// TwinCAT 3 PLC project PLC_UU_V01
// ProgramVersion: 3.1.4022.4
// libraries:
//   Tc2_MC2, * (Beckhoff Automation GmbH)
//   Tc2_Standard, * (Beckhoff Automation GmbH)
//   Tc2_System, * (Beckhoff Automation GmbH)
//   Tc3_Module, * (Beckhoff Automation GmbH)
//   VisuDialogs, * (System)
// project tree:
//   DUTs/ ST_AxisIn.TcDUT, ST_AxisInterface.TcDUT, ST_AxisOut.TcDUT, ST_Demo.TcDUT
//   / GlobalTextList.TcGTLO, PlcTask.TcTTO, Visualization Manager.TcVMO (not stored)
//   GVLs/ GVL_IO.TcGVL, GVL_Servo.TcGVL
//   POUs/ FB_Motion.TcPOU, MAIN.TcPOU, PRG_Servo1.TcPOU
//   VISUs/ TC_SERVO1.TcVIS

CONFIGURATION PLC_UU_V01
    RESOURCE PLC ON TwinCAT3
        TASK PlcTask(INTERVAL := T#10ms, PRIORITY := 20);
        PROGRAM MAIN WITH PlcTask : MAIN;
    END_RESOURCE
END_CONFIGURATION

// ---- DUTs/ST_AxisIn.TcDUT
TYPE ST_AxisIn :
STRUCT
	bEnable		: BOOL;
	fOverride	: LREAL;
	bManuelFw	: BOOL;
	bManuelBw	: BOOL;
	fVelocity	: LREAL;
	bMoveAbs	: BOOL;
	fPosition	: LREAL;
	bStop		:BOOL;
	bReset		:BOOL;

END_STRUCT
END_TYPE

// ---- DUTs/ST_AxisInterface.TcDUT
TYPE ST_AxisInterface :
STRUCT
	INPUT	: ST_AxisIn;
	OUTPUT	: ST_AxisOut;
	
END_STRUCT
END_TYPE

// ---- DUTs/ST_AxisOut.TcDUT
TYPE ST_AxisOut :
STRUCT
	bEnabled	: BOOL;
	bJogBusy	: BOOL;
	bJogDone	: BOOL;
	bMoveAbsDone: BOOL;
	bMoveAbsBusy: BOOL;
	bJogError	: BOOL;
	bPowerErr	: BOOL;
	bMoveAbsErr	: BOOL;
	bStopDone	: BOOL;
	bStopBusy	: BOOL;
	bStopErr	: BOOL;
	bStopActive : BOOL;	
	bResetDone	:BOOL;

END_STRUCT
END_TYPE

// ---- DUTs/ST_Demo.TcDUT
TYPE ST_Demo :
STRUCT
	bVar	: BOOL;
	sVar	: STRING;
	nVar	: INT;
	fVar	: LREAL;
	
END_STRUCT
END_TYPE

// ---- GVLs/GVL_IO.TcGVL
VAR_GLOBAL
	bInput1	AT%I*	: BOOL;
	bInput2	AT%I*	: BOOL;
	bInput3	AT%I*	: BOOL;
	bInput4	AT%I*	: BOOL;
	
	bOutput1	AT%Q*	: BOOL;
	bOutput2	AT%Q*	: BOOL;
	bOutput3	AT%Q*	: BOOL;
	bOutput4	AT%Q*	: BOOL;
	
	nInput1		AT%I*	: INT;
	nInput2		AT%I*	: INT;
	
	nOutput1	AT%Q*	: INT;
	nOutput2	AT%Q*	: INT;
	
END_VAR

// ---- GVLs/GVL_Servo.TcGVL
VAR_GLOBAL
	Axis1	: AXIS_REF;
	Axis2	: AXIS_REF;
	
	stAxis1	: ST_AxisInterface;
	stAxis2	: ST_AxisInterface;
	
	fbMotion1	: FB_Motion;
	fbMotion2	: FB_Motion;
	
END_VAR

// ---- POUs/MAIN.TcPOU
PROGRAM MAIN
VAR
	stDemo	: ST_Demo;
	stArrayDemo	: ARRAY[1..100]OF ST_Demo;
	
	i: INT;
	
END_VAR

IF bInput1	THEN
	FOR i:= 0 TO 100 DO
		stArrayDemo[i+1].nVar	:= i*i;
		stArrayDemo[i+1].fVar	:= INT_TO_LREAL(i)+1.345;
	END_FOR
END_IF

ACT_Motion();

PRG_Servo1();

ACTION ACT_Motion:
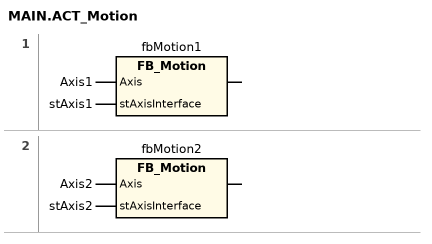
// NETWORK 1
fbMotion1(Axis := Axis1, stAxisInterface := stAxis1); // FB_Motion

// NETWORK 2
fbMotion2(Axis := Axis2, stAxisInterface := stAxis2); // FB_Motion
END_ACTION

END_PROGRAM

// ---- POUs/PRG_Servo1.TcPOU
PROGRAM PRG_Servo1
VAR
	nState: INT;
	bBaslat	: bool;
	bSensor1: BOOL;
	rSayici: R_TRIG;
	bSensor2: BOOL;
	nSayici: INT;
	nCounter: INT;
END_VAR

stAxis1.INPUT.bEnable	:= TRUE;
staxis1.INPUT.bStop:=FALSE;
stAxis1.INPUT.bReset := FALSE;


rSayici(CLK:= bSensor2, Q=> );
CASE nState OF
	
0:
	IF bBaslat AND staxis1.OUTPUT.bEnabled AND NOT stAxis1.OUTPUT.bPowerErr THEN
		nState	:= 10;
		nCounter := 0;
	END_IF
	
10:
	stAxis1.INPUT.bMoveAbs	:= TRUE;
	stAxis1.INPUT.fVelocity	:= 4000;
	stAxis1.INPUT.fPosition	:= 30000;
	
	IF stAxis1.OUTPUT.bMoveAbsBusy AND NOT stAxis1.OUTPUT.bMoveAbsErr THEN

		nState					:= 20;
		stAxis1.INPUT.bMoveAbs:=FALSE;

	ELSIF stAxis1.OUTPUT.bMoveAbsErr THEN
	
	nState					:= 999;
	nCounter := nState;
	stAxis1.INPUT.bMoveAbs	:= FALSE;

	END_IF
			
20:
	IF stAxis1.OUTPUT.bMoveAbsDone AND NOT stAxis1.OUTPUT.bMoveAbsErr THEN
		nState					:= 30;
		nCounter := nState;

	ELSIF stAxis1.OUTPUT.bMoveAbsErr THEN	
		nState					:= 999;
		nCounter := nState;

	END_IF
	
30:	
	IF bSensor1 THEN
		nState	:= 40;
		nCounter:=nState;
	END_IF
	
40:
	nCounter:=30;

	stAxis1.INPUT.bMoveAbs	:= TRUE;
	stAxis1.INPUT.fVelocity	:= 7000;
	stAxis1.INPUT.fPosition	:= 50000;
	
	IF stAxis1.OUTPUT.bMoveAbsBusy AND NOT stAxis1.OUTPUT.bMoveAbsErr THEN
		stAxis1.INPUT.bMoveAbs	:= FALSE;
		nState					:= 50;

	ELSIF stAxis1.OUTPUT.bMoveAbsErr THEN
		nState					:= 999;
		nCounter := nState;

		stAxis1.INPUT.bMoveAbs	:= FALSE;		
	END_IF
	
50:
	IF stAxis1.OUTPUT.bMoveAbsDone AND NOT stAxis1.OUTPUT.bMoveAbsErr THEN
		nState					:= 60;
		nCounter := nState;

	ELSIF stAxis1.OUTPUT.bMoveAbsErr THEN	
		nState					:= 999;
		nCounter := nState;

	END_IF

60:
	IF rSayici.Q AND nSayici<5 THEN
		nSayici	:= nSayici+1;	
	ELSIF nSayici>=5 THEN
		nSayici	:=0;
		nState	:= 70;
		nCounter := nState;
	END_IF

70:
	stAxis1.INPUT.bMoveAbs	:= TRUE;

	stAxis1.INPUT.fVelocity	:= 8000;
	stAxis1.INPUT.fPosition	:= 0;
	nCounter:=60;
	IF stAxis1.OUTPUT.bMoveAbsBusy AND NOT stAxis1.OUTPUT.bMoveAbsErr THEN
		stAxis1.INPUT.bMoveAbs	:= FALSE;
		nState					:= 80;
		nCounter := nState;

	ELSIF stAxis1.OUTPUT.bMoveAbsErr THEN
		nState					:= 999;
		nCounter := nState;

		stAxis1.INPUT.bMoveAbs	:= FALSE;		
	END_IF
	
80:
	IF stAxis1.OUTPUT.bMoveAbsDone AND NOT stAxis1.OUTPUT.bMoveAbsErr THEN
				nState	:= 0;
				nCounter := nState;

	ELSIF stAxis1.OUTPUT.bMoveAbsErr THEN	
		nState					:= 999;
		nCounter := nState;

	END_IF
	
END_CASE

IF stAxis1.OUTPUT.bPowerErr THEN
	stAxis1.INPUT.bReset := TRUE;
	nState:=0;
END_IF

IF NOT bBaslat THEN
	
staxis1.INPUT.bStop:=TRUE;
stAxis1.INPUT.bMoveAbs	:= FALSE;
staxis1.OUTPUT.bEnabled:=TRUE;


		IF staxis1.OUTPUT.bEnabled
		AND NOT stAxis1.OUTPUT.bPowerErr 
		AND NOT stAxis1.OUTPUT.bMoveAbsErr
		AND NOT staxis1.OUTPUT.bStopErr 
		AND  staxis1.OUTPUT.bStopBusy THEN
	
	staxis1.INPUT.bStop:=FALSE;
	nState:=nCounter;

	END_IF

END_IF

END_PROGRAM

// ---- POUs/FB_Motion.TcPOU
FUNCTION_BLOCK FB_Motion
VAR_INPUT

	
END_VAR
VAR_OUTPUT
	
END_VAR
VAR
	fbMcPower	: MC_Power;
	fbMcJog: MC_Jog;
	fbMcMoveAbs: MC_MoveAbsolute;
	fbMcStop: MC_Stop;
	fbMcReset: MC_Reset;
END_VAR

VAR_IN_OUT
	Axis			: AXIS_REF;
	stAxisInterface	: ST_AxisInterface;
	
END_VAR

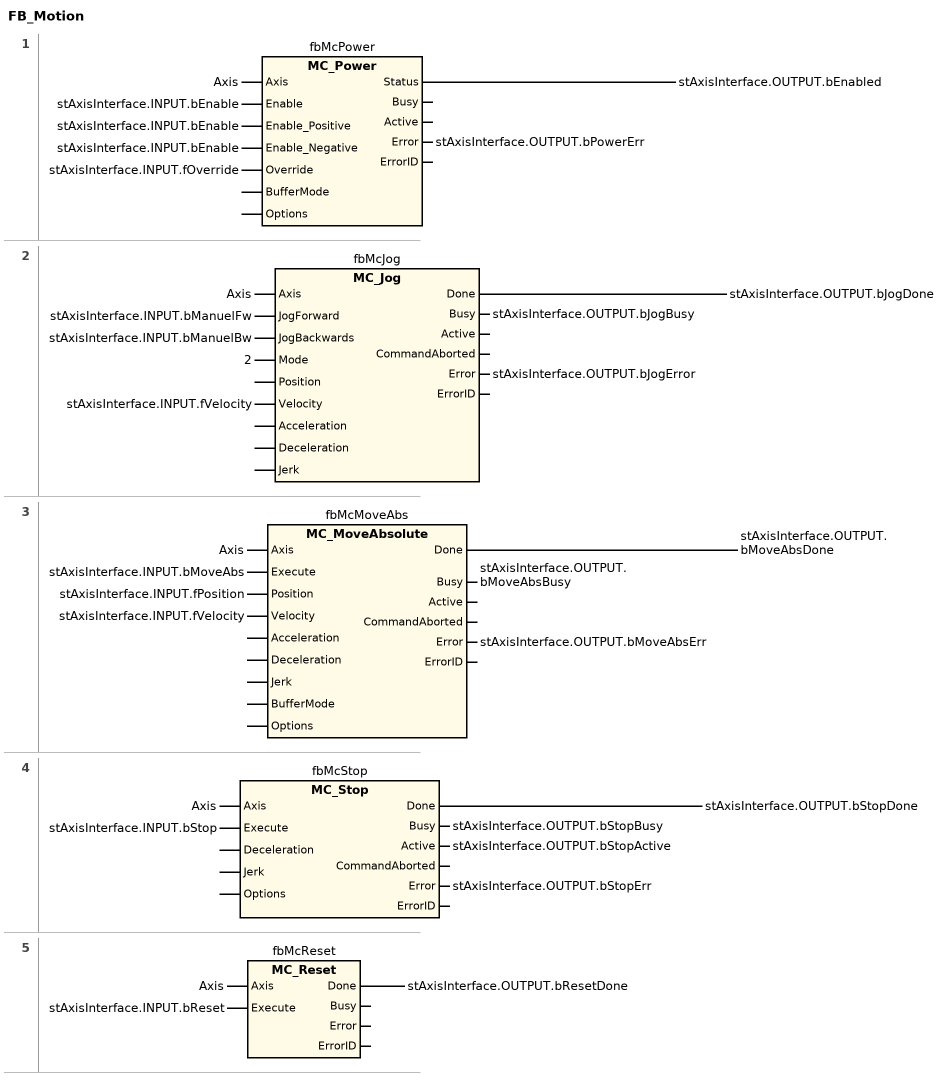
// NETWORK 1
fbMcPower(
    Axis := Axis,
    Enable := stAxisInterface.INPUT.bEnable,
    Enable_Positive := stAxisInterface.INPUT.bEnable,
    Enable_Negative := stAxisInterface.INPUT.bEnable,
    Override := stAxisInterface.INPUT.fOverride,
    Error => stAxisInterface.OUTPUT.bPowerErr); // MC_Power
stAxisInterface.OUTPUT.bEnabled := fbMcPower.Status;

// NETWORK 2
fbMcJog(
    Axis := Axis,
    JogForward := stAxisInterface.INPUT.bManuelFw,
    JogBackwards := stAxisInterface.INPUT.bManuelBw,
    Mode := 2,
    Velocity := stAxisInterface.INPUT.fVelocity,
    Busy => stAxisInterface.OUTPUT.bJogBusy,
    Error => stAxisInterface.OUTPUT.bJogError); // MC_Jog
stAxisInterface.OUTPUT.bJogDone := fbMcJog.Done;

// NETWORK 3
fbMcMoveAbs(
    Axis := Axis,
    Execute := stAxisInterface.INPUT.bMoveAbs,
    Position := stAxisInterface.INPUT.fPosition,
    Velocity := stAxisInterface.INPUT.fVelocity,
    Busy => stAxisInterface.OUTPUT.bMoveAbsBusy,
    Error => stAxisInterface.OUTPUT.bMoveAbsErr); // MC_MoveAbsolute
stAxisInterface.OUTPUT.bMoveAbsDone := fbMcMoveAbs.Done;

// NETWORK 4
fbMcStop(
    Axis := Axis,
    Execute := stAxisInterface.INPUT.bStop,
    Busy => stAxisInterface.OUTPUT.bStopBusy,
    Active => stAxisInterface.OUTPUT.bStopActive,
    Error => stAxisInterface.OUTPUT.bStopErr); // MC_Stop
stAxisInterface.OUTPUT.bStopDone := fbMcStop.Done;

// NETWORK 5
fbMcReset(Axis := Axis, Execute := stAxisInterface.INPUT.bReset); // MC_Reset
stAxisInterface.OUTPUT.bResetDone := fbMcReset.Done;

END_FUNCTION_BLOCK

// ---- GlobalTextList.TcGTLO
TEXTLIST GlobalTextList
  587 = '%.1f'
  538 = '%f'
  929 = 'ABS BUSY'
  664 = 'ACT POS'
  475 = 'ACT VELO'
  733 = 'MANUEL BUSY'
  93 = 'MOTOR ENABLE'
  245 = 'SET POS'
  591 = 'SET VELO'
END_TEXTLIST

// ---- VISUs/TC_SERVO1.TcVIS
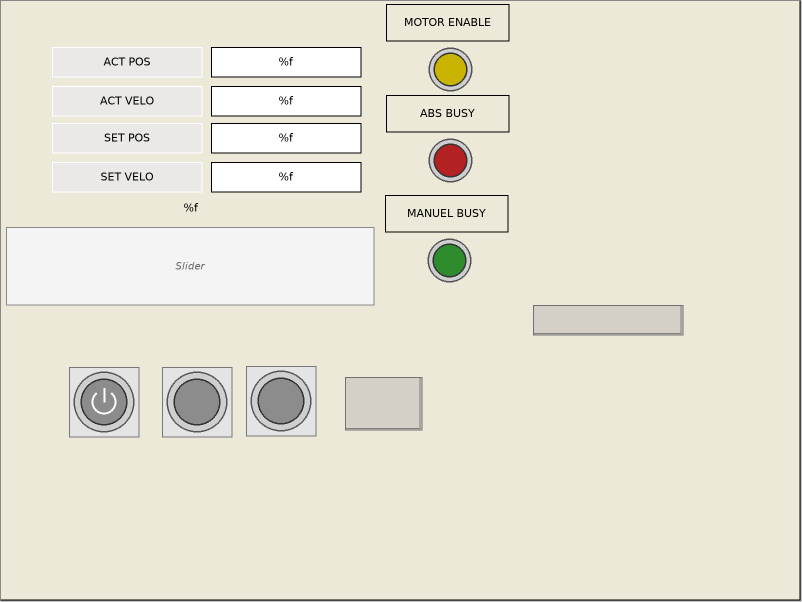
VISUALIZATION TC_SERVO1  // 802x602
    Rectangle (0,0 800x600)
    Rectangle (52,47 150x30), "ACT POS"
    Rectangle (211,47 150x30), "%f", text variable: Axis1.NcToPlc.ActPos
    Rectangle (52,86 150x30), "ACT VELO"
    Rectangle (211,86 150x30), "%f", text variable: Axis1.NcToPlc.ActVelo
    Rectangle (52,123 150x30), "SET POS"
    Rectangle (211,123 150x30), "%f", text variable: MAIN.fPos1
        OnMouseClick: write the text variable via VisuDialogs.Numpad
    Rectangle (52,162 150x30), "SET VELO"
    Rectangle (211,162 150x30), "%f", text variable: MAIN.fVelocity1
        OnMouseClick: write the text variable via VisuDialogs.Numpad
    Slider (6,227 368x78), variable: MAIN.fOverride1, scale 0..100
    Rectangle (160,194 62x28), "%f", text variable: MAIN.fOverride1
    PowerSwitch (69,367 70x70), variable: MAIN.bEnable1, behaviour: TOGGLE, style: Switch-PowerSwitch-Gray
    PushSwitch (162,367 70x70), variable: MAIN.bManuelBw1, behaviour: TOGGLE, style: Switch-PushSwitch-Gray
    PushSwitch (246,366 70x70), variable: MAIN.bManuelFw1, behaviour: TOGGLE, style: Switch-PushSwitch-Gray
    Button (345,377 77x53)
        tap MAIN.bMoveAbs1
    Lamp1 (424,44 53x51), variable: MAIN.bEnabled1, style: Lamp-Lamp1-Yellow
    Rectangle (386,4 123x37), "MOTOR ENABLE"
    Lamp1 (424,135 53x51), variable: MAIN.bMoveAbsBusy1, style: Lamp-Lamp1-Red
    Rectangle (386,95 123x37), "ABS BUSY"
    Lamp1 (423,235 53x51), variable: MAIN.bJogBusy1, style: Lamp-Lamp1-Green
    Rectangle (385,195 123x37), "MANUEL BUSY"
    Button (533,305 150x30)
END_VISUALIZATION
